FUNCTION_BLOCK Section0Ctrl
  (* Standard: 61499-2 *)
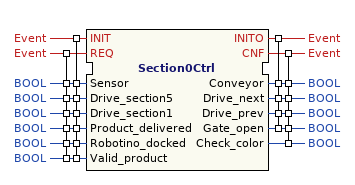
  EVENT_INPUT
    INIT WITH Sensor, Drive_section5, Drive_section1, Product_delivered, Robotino_docked, Valid_product;
    REQ WITH Sensor, Drive_section5, Drive_section1, Product_delivered, Robotino_docked, Valid_product;
  END_EVENT
  EVENT_OUTPUT
    INITO WITH Conveyor, Drive_next, Drive_prev, Gate_open;
    CNF WITH Conveyor, Drive_next, Drive_prev, Gate_open, Check_color;
  END_EVENT
  VAR_INPUT
    Sensor : BOOL;
    Drive_section5 : BOOL;
    Drive_section1 : BOOL;
    Product_delivered : BOOL;
    Robotino_docked : BOOL;
    Valid_product : BOOL;
  END_VAR
  VAR_OUTPUT
    Conveyor : BOOL;
    Drive_next : BOOL;
    Drive_prev : BOOL;
    Gate_open : BOOL;
    Check_color : BOOL;
  END_VAR
  VAR
    TimeStamp : DATE_AND_TIME;
  END_VAR
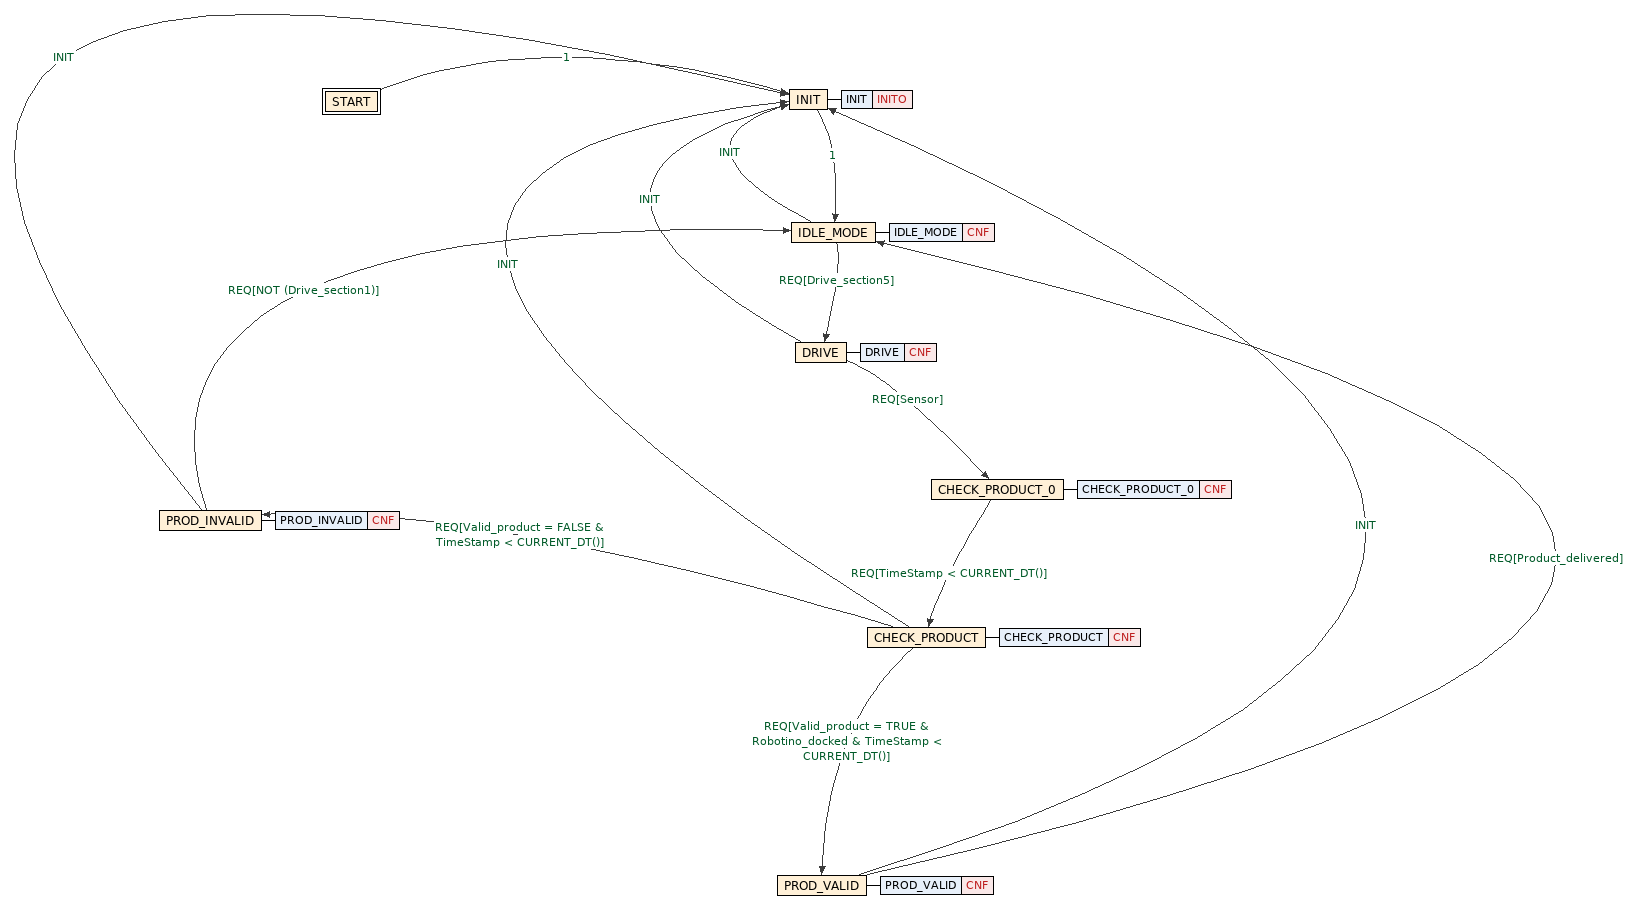
  EC_STATES
    START;
    INIT : INIT -> INITO;
    IDLE_MODE : IDLE_MODE -> CNF;
    DRIVE : DRIVE -> CNF;
    CHECK_PRODUCT : CHECK_PRODUCT -> CNF;
    PROD_VALID : PROD_VALID -> CNF;
    PROD_INVALID : PROD_INVALID -> CNF;
    CHECK_PRODUCT_0 : CHECK_PRODUCT_0 -> CNF;
  END_STATES
  EC_TRANSITIONS
    START TO INIT := 1;
    INIT TO IDLE_MODE := 1;
    IDLE_MODE TO INIT := INIT;
    IDLE_MODE TO DRIVE := REQ[Drive_section5];
    DRIVE TO INIT := INIT;
    DRIVE TO CHECK_PRODUCT_0 := REQ[Sensor];
    CHECK_PRODUCT TO INIT := INIT;
    CHECK_PRODUCT TO PROD_VALID := REQ[Valid_product = TRUE & Robotino_docked & TimeStamp < CURRENT_DT()];
    CHECK_PRODUCT TO PROD_INVALID := REQ[Valid_product = FALSE & TimeStamp < CURRENT_DT()];
    PROD_VALID TO INIT := INIT;
    PROD_INVALID TO INIT := INIT;
    PROD_INVALID TO IDLE_MODE := REQ[NOT (Drive_section1)];
    PROD_VALID TO IDLE_MODE := REQ[Product_delivered];
    CHECK_PRODUCT_0 TO CHECK_PRODUCT := REQ[TimeStamp < CURRENT_DT()];
  END_TRANSITIONS
  ALGORITHM INIT IN ST:
Conveyor := FALSE;&#10;Gate_open := FALSE;&#10;Drive_prev := FALSE;&#10;Drive_next := FALSE;&#10;
  END_ALGORITHM
  ALGORITHM IDLE_MODE IN ST:
Conveyor := FALSE;&#10;Gate_open := FALSE;&#10;Drive_prev := TRUE;&#10;Drive_next := FALSE;&#10;Check_color := FALSE;&#10;
  END_ALGORITHM
  ALGORITHM DRIVE IN ST:
Conveyor := TRUE;&#10;Gate_open := FALSE;&#10;Drive_prev := TRUE;&#10;Drive_next := FALSE;&#10;
  END_ALGORITHM
  ALGORITHM CHECK_PRODUCT IN ST:
Conveyor := FALSE;&#10;Gate_open := FALSE;&#10;Drive_prev := FALSE;&#10;Drive_next := FALSE;&#10;Check_color := TRUE;&#10;TimeStamp := ADD_DT_TIME(CURRENT_DT());&#10;
  END_ALGORITHM
  ALGORITHM PROD_VALID IN ST:
Conveyor := TRUE;&#10;Gate_open := TRUE;&#10;Drive_prev := FALSE;&#10;Drive_next := FALSE;&#10;
  END_ALGORITHM
  ALGORITHM PROD_INVALID IN ST:
Conveyor := TRUE;&#10;Gate_open := FALSE;&#10;Drive_prev := FALSE;&#10;Drive_next := TRUE;&#10;
  END_ALGORITHM
  ALGORITHM CHECK_PRODUCT_0 IN ST:
Conveyor := FALSE;&#10;Gate_open := FALSE;&#10;Drive_prev := FALSE;&#10;Drive_next := FALSE;&#10;Check_color := TRUE;&#10;TimeStamp := ADD_DT_TIME(CURRENT_DT());&#10;
  END_ALGORITHM
END_FUNCTION_BLOCK
